FUNCTION_BLOCK fb_motionController
VAR_INPUT
	in_flg_run : BOOL;
END_VAR
VAR_OUTPUT
	out_flg_run : BOOL;
END_VAR
VAR_IN_OUT
	var_ref_X : ref_mc_moveAbs;
	var_ref_Y : ref_mc_moveAbs;
	var_ref_Z : ref_mc_moveAbs;
END_VAR
VAR_INPUT
	in_flg_start : BOOL;
	in_var_targetPosX : LREAL;
	in_var_targetPosY : LREAL;
	in_var_targetPosZ : LREAL;
	in_var_direction : eP_motionDirection;
	
END_VAR
VAR_OUTPUT
	out_flg_busy : BOOL;
	out_flg_Done : BOOL;
	out_flg_moveXYDone : BOOL;
	
END_VAR
VAR
	SFCInit : BOOL;
	fbi_r_TIRG: R_TRIG;
	fbi_f_TRIG: F_TRIG;
	var_buf_targetPosX: LREAL;
	var_buf_targetPosY: LREAL;
	var_buf_targetPosZ: LREAL;
	var_buf_direction: eP_motionDirection;
	trn_getParamDone: BOOL;
	var_mutex: INT;
	trn_moveXY_1Done: BOOL;
	trn_moveZ_1Done: BOOL;
	trn_moveZ_2Done: BOOL;
	trn_moveXY_2Done: BOOL;
	
	trn_moveX_3Done: BOOL;
	trn_moveY_3Done: BOOL;
	trn_moveZ_3Done: BOOL;
	
	trn_moveX_4Done: BOOL;
	trn_moveY_4Done: BOOL;
	trn_moveZ_4Done: BOOL;

	trn_executeReset2Done: BOOL;
	var_process: INT;
END_VAR

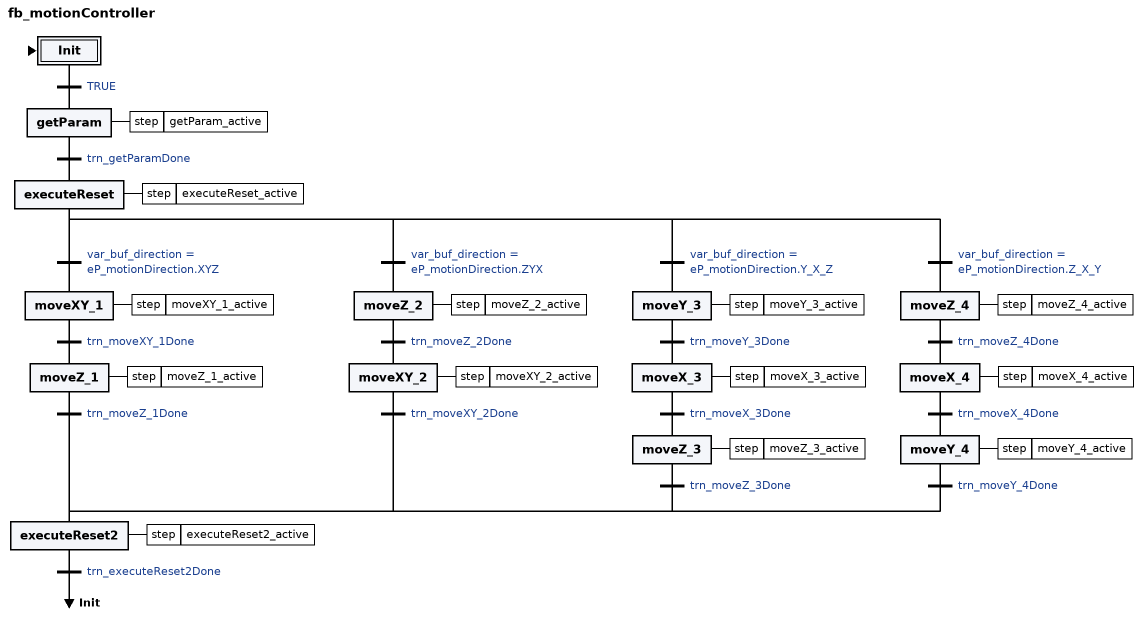
INITIAL_STEP Init:
END_STEP
TRANSITION FROM Init TO getParam
    := TRUE;
END_TRANSITION
STEP getParam:
    getParam_active(N);  // step action
END_STEP
TRANSITION FROM getParam TO executeReset
    := trn_getParamDone;
END_TRANSITION
STEP executeReset:
    executeReset_active(N);  // step action
END_STEP
TRANSITION FROM executeReset TO moveXY_1
    := var_buf_direction = eP_motionDirection.XYZ;
END_TRANSITION
STEP moveXY_1:
    moveXY_1_active(N);  // step action
END_STEP
TRANSITION FROM moveXY_1 TO moveZ_1
    := trn_moveXY_1Done;
END_TRANSITION
STEP moveZ_1:
    moveZ_1_active(N);  // step action
END_STEP
TRANSITION FROM moveZ_1 TO executeReset2
    := trn_moveZ_1Done;
END_TRANSITION
TRANSITION FROM executeReset TO moveZ_2
    := var_buf_direction = eP_motionDirection.ZYX;
END_TRANSITION
STEP moveZ_2:
    moveZ_2_active(N);  // step action
END_STEP
TRANSITION FROM moveZ_2 TO moveXY_2
    := trn_moveZ_2Done;
END_TRANSITION
STEP moveXY_2:
    moveXY_2_active(N);  // step action
END_STEP
TRANSITION FROM moveXY_2 TO executeReset2
    := trn_moveXY_2Done;
END_TRANSITION
TRANSITION FROM executeReset TO moveY_3
    := var_buf_direction = eP_motionDirection.Y_X_Z;
END_TRANSITION
STEP moveY_3:
    moveY_3_active(N);  // step action
END_STEP
TRANSITION FROM moveY_3 TO moveX_3
    := trn_moveY_3Done;
END_TRANSITION
STEP moveX_3:
    moveX_3_active(N);  // step action
END_STEP
TRANSITION FROM moveX_3 TO moveZ_3
    := trn_moveX_3Done;
END_TRANSITION
STEP moveZ_3:
    moveZ_3_active(N);  // step action
END_STEP
TRANSITION FROM moveZ_3 TO executeReset2
    := trn_moveZ_3Done;
END_TRANSITION
TRANSITION FROM executeReset TO moveZ_4
    := var_buf_direction = eP_motionDirection.Z_X_Y;
END_TRANSITION
STEP moveZ_4:
    moveZ_4_active(N);  // step action
END_STEP
TRANSITION FROM moveZ_4 TO moveX_4
    := trn_moveZ_4Done;
END_TRANSITION
STEP moveX_4:
    moveX_4_active(N);  // step action
END_STEP
TRANSITION FROM moveX_4 TO moveY_4
    := trn_moveX_4Done;
END_TRANSITION
STEP moveY_4:
    moveY_4_active(N);  // step action
END_STEP
TRANSITION FROM moveY_4 TO executeReset2
    := trn_moveY_4Done;
END_TRANSITION
STEP executeReset2:
    executeReset2_active(N);  // step action
END_STEP
TRANSITION FROM executeReset2 TO Init
    := trn_executeReset2Done;
END_TRANSITION

ACTION executeReset_active:
IF executeReset._x AND executeReset.x = FALSE THEN
	var_ref_x.Execute := FALSE;
	var_ref_y.Execute := FALSE;
	var_ref_z.Execute := FALSE;
ELSIF executeReset._x AND executeReset.x THEN
	var_ref_x.Execute := FALSE;
	var_ref_y.Execute := FALSE;
	var_ref_z.Execute := FALSE;
END_IF
END_ACTION

ACTION executeReset2_active:
IF executeReset2._x AND executeReset2.x= FALSE THEN
	trn_executeReset2Done := FALSE;
	var_ref_x.Execute := FALSE;
	var_ref_y.Execute := FALSE;
	var_ref_z.Execute := FALSE;
	out_flg_done := TRUE;
	out_flg_moveXYDone := FALSE;
ELSIF executeReset2._x AND executeReset2.x THEN
	var_ref_x.Execute := FALSE;
	var_ref_y.Execute := FALSE;
	var_ref_z.Execute := FALSE;
	trn_executeReset2Done := TRUE;
	out_flg_done := FALSE;
	in_flg_start := FALSE;
END_IF
END_ACTION

ACTION getParam_active:
fbi_r_TIRG(CLK:= in_flg_start, Q=> );
IF getParam._x AND getParam.x = FALSE THEN
	var_mutex := 0;
	trn_getParamDone := FALSE;
	out_flg_moveXYDone:= FALSE;
	in_flg_start := FALSE;
ELSIF getParam._x AND getParam.x THEN
	IF fbi_r_TIRG.Q THEN
		var_ref_x.Position := in_var_targetPosX;
		var_ref_Y.Position := in_var_targetPosY;
		var_ref_Z.Position := in_var_targetPosZ;
		var_buf_direction := in_var_direction;
		var_mutex := 1;
	END_IF
	IF var_mutex = 1 THEN
		out_flg_busy := TRUE;
		trn_getParamDone := TRUE;
	ELSE
		out_flg_busy := FALSE;
		trn_getParamDone := FALSE;
	END_IF
	IF in_flg_run THEN
		out_flg_run := TRUE;
	ELSE
		out_flg_run := FALSE;
	END_IF
END_IF
END_ACTION

ACTION moveX_3_active:
IF moveX_3._x AND moveX_3.x = FALSE THEN
	trn_moveX_3Done := FALSE;
	var_process := 0;
ELSIF moveX_3._x AND moveX_3.x THEN
	CASE var_process OF
		0:
			var_ref_x.Execute := TRUE;
			var_process := 1;
		1:
			IF var_ref_x.Done THEN
				trn_moveX_3Done := TRUE;
			END_IF
	END_CASE
END_IF
END_ACTION

ACTION moveX_4_active:
IF moveX_4._x AND moveX_4.x = FALSE THEN
	trn_moveX_4Done := FALSE;
	var_process := 0;
ELSIF moveX_4._x AND moveX_4.x THEN
	CASE var_process OF
		0:
			var_ref_x.Execute := TRUE;
			var_process := 1;
		1:
			IF var_ref_x.Done THEN
				trn_moveX_4Done := TRUE;
			END_IF
	END_CASE
END_IF
END_ACTION

ACTION moveXY_1_active:
IF moveXY_1._x AND moveXY_1.x = FALSE THEN
	out_flg_moveXYDone:= FALSE;
	trn_moveXY_1Done := FALSE;
	var_process := 0;
ELSIF moveXY_1._x AND moveXY_1.x THEN
	CASE var_process OF
		0:
			var_ref_x.Execute := TRUE;
			var_ref_y.Execute := TRUE;
			var_process := 1;
		1:
			IF var_ref_x.Done AND var_ref_y.Done THEN
				out_flg_moveXYDone:= TRUE;
				trn_moveXY_1Done := TRUE;
			END_IF
	END_CASE
END_IF
END_ACTION

ACTION moveXY_2_active:
IF moveXY_2._x AND moveXY_2.x = FALSE THEN
	trn_moveXY_2Done := FALSE;
	var_process := 0;
ELSIF moveXY_2._x AND moveXY_2.x THEN
	CASE var_process OF
		0:
			var_ref_x.Execute := TRUE;
			var_ref_y.Execute := TRUE;
			var_process := 1;
		1:
			IF var_ref_x.Done AND var_ref_y.Done THEN
				trn_moveXY_2Done := TRUE;
			END_IF
	END_CASE
END_IF
END_ACTION

ACTION moveY_3_active:
IF moveY_3._x AND moveY_3.x = FALSE THEN
	trn_moveY_3Done := FALSE;
	var_process := 0;
ELSIF moveY_3._x AND moveY_3.x THEN
	CASE var_process OF
		0:
			var_ref_y.Execute := TRUE;
			var_process := 1;
		1:
			IF var_ref_y.Done THEN
				trn_moveY_3Done := TRUE;
			END_IF
	END_CASE
END_IF
END_ACTION

ACTION moveY_4_active:
IF moveY_4._x AND moveY_4.x = FALSE THEN
	trn_moveY_4Done := FALSE;
	var_process := 0;
ELSIF moveY_4._x AND moveY_4.x THEN
	CASE var_process OF
		0:
			var_ref_y.Execute := TRUE;
			var_process := 1;
		1:
			IF var_ref_y.Done THEN
				trn_moveY_4Done := TRUE;
			END_IF
	END_CASE
END_IF
END_ACTION

ACTION moveZ_1_active:
IF moveZ_1._x AND moveZ_1.x = FALSE THEN
	out_flg_moveXYDone := FALSE;
	trn_moveZ_1Done := FALSE;
	var_process := 0;
ELSIF moveZ_1._x AND moveZ_1.x THEN
	CASE var_process OF
		0:
			var_ref_z.Execute := TRUE;
			var_process := 1;
		1:
			IF var_ref_z.Done THEN
				trn_moveZ_1Done := TRUE;
			END_IF
	END_CASE
	

END_IF
END_ACTION

ACTION moveZ_2_active:
IF moveZ_2._x AND moveZ_2.x = FALSE THEN
	trn_moveZ_2Done := FALSE;
	var_process := 0;
ELSIF moveZ_2._x AND moveZ_2.x THEN
	CASE var_process OF
		0:
			var_ref_z.Execute := TRUE;
			var_process := 1;
		1:
			IF var_ref_z.Done THEN
				trn_moveZ_2Done := TRUE;
			END_IF
	END_CASE
END_IF
END_ACTION

ACTION moveZ_3_active:
IF moveZ_3._x AND moveZ_3.x = FALSE THEN
	trn_moveZ_3Done := FALSE;
	var_process := 0;
ELSIF moveZ_3._x AND moveZ_3.x THEN
	CASE var_process OF
		0:
			var_ref_Z.Execute := TRUE;
			var_process := 1;
		1:
			IF var_ref_Z.Done THEN
				trn_moveZ_3Done := TRUE;
			END_IF
	END_CASE
END_IF
END_ACTION

ACTION moveZ_4_active:
IF moveZ_4._x AND moveZ_4.x = FALSE THEN
	trn_moveZ_4Done := FALSE;
	var_process := 0;
ELSIF moveZ_4._x AND moveZ_4.x THEN
	CASE var_process OF
		0:
			var_ref_z.Execute := TRUE;
			var_process := 1;
		1:
			IF var_ref_z.Done THEN
				trn_moveZ_4Done := TRUE;
			END_IF
	END_CASE
END_IF
END_ACTION

PROPERTY p_Init : bool
GET
p_init := THIS^.SFCInit;
END_GET
SET
THIS^.SFCInit := p_init;
END_SET
END_PROPERTY

END_FUNCTION_BLOCK

(* stored: Version 1.1.0.1, ProductVersion 3.1.4024.11
   POU fb_motionController: Id {52e806b7-7190-4076-b358-348a2951a77d}, SpecialFunc None
   Action executeReset_active: Id {26f49e73-44db-4ad6-96a9-4a3452650bcc}
   Action executeReset2_active: Id {2e0f8b94-1d1f-45df-8449-27ab46ddcc95}
   Action getParam_active: Id {ca87f63c-b54a-4baf-9969-231a0f0889a6}
   Action moveX_3_active: Id {173ff45e-bb0d-4fb7-989c-6546ec05051f}
   Action moveX_4_active: Id {59c11aa8-af24-40f7-85e3-90df7ac6893e}
   Action moveXY_1_active: Id {b4647fdb-7b43-4b39-927c-694ce7770750}
   Action moveXY_2_active: Id {5249e92d-0fb2-4377-8fb4-15d46b95658f}
   Action moveY_3_active: Id {8ddec246-2e1f-4814-aa9c-f5e45a39efde}
   Action moveY_4_active: Id {e447f6e9-794c-4431-8308-39a858c11129}
   Action moveZ_1_active: Id {25d1b2ee-857b-4a4b-8b6b-1ab83cb3af47}
   Action moveZ_2_active: Id {4208bc77-ecd8-49be-801d-08cb671f2412}
   Action moveZ_3_active: Id {580e6cfe-f417-4cfd-943d-7a3195951506}
   Action moveZ_4_active: Id {424b7113-3562-45de-ab82-430cce7c804a}
   Property p_Init: Id {a40cea0f-dc73-4847-92e9-3de4325c2127}
   Get Get: Id {c05d407d-75eb-491d-8513-de4cb6a9bdd1}
   Set Set: Id {759c94c9-33f6-4682-9919-b55424a280ac} *)
